// TwinCAT 3 PLC project Untitled1_1
// ProgramVersion: 3.1.4024.0
// libraries:
//   Tc2_MC2, * (Beckhoff Automation GmbH)
//   Tc2_Standard, * (Beckhoff Automation GmbH)
//   Tc2_System, * (Beckhoff Automation GmbH)
//   Tc2_Utilities, * (Beckhoff Automation GmbH)
//   Tc3_IotBase, * (Beckhoff Automation GmbH)
//   Tc3_JsonXml, * (Beckhoff Automation GmbH)
//   Tc3_Module, * (Beckhoff Automation GmbH)
// project tree:
//   DUTs/ E_Mode.TcDUT, E_State.TcDUT, ST_jsoncmd.TcDUT
//   / GlobalTextList.TcGTLO, PlcTask.TcTTO, Visualization Manager.TcVMO (not stored)
//   GVLs/ Comms.TcGVL, E_HomeState.TcDUT, E_LifterState.TcDUT, IO.TcGVL, Slots.TcGVL, ST_Coord.TcDUT, ST_Message.TcDUT
//   POUs/ FBMotion.TcPOU, FB_Lifter.TcPOU, MAIN.TcPOU, Motion.TcPOU, MqttClient.TcPOU, PrgMqttCom.TcPOU
//   VISUs/ Visualization.TcVIS
// real-time tasks:
//   TASK PlcTask: cycle T#10ms, priority 20, ADS port 350
// motion (NC):
//   TASK NC-Task 1 SAF: cycle T#2ms, priority 4, ADS port 501
//   TASK NC-Task 1 SVB: cycle T#10ms, priority 8, ADS port 511
//   AXIS Axis 1 (id 1)
//     Dynamic: Acceleration=322.5, Deceleration=322.5, Jerk=7172.84
//     Velo: SlowManual=10, FastManual=50, Maximum=50
//     OtherSettings: AllowMotionCmdToSlave=true
//     encoder EncType=19
//       EncPara: ScaleFactorNumerator=0.00086, MaxCount=#xffffffff
//     drive DrvType=16
//       DrvPara: MaxCount=#xffffffff, DriveControlDWord=#x00020100
//         Analog: VeloReferenz=50, TorqueSetpointScale=10, ScaleFactorActTorque=0.1
//         TimeComp: TaskDelayCycles=1
//     controller CtrType=1
//       CtrPara: PriorControlFactor=1
//         Observer: BandWidth=20
//   AXIS Axis 2 (id 2)
//     Dynamic: Acceleration=330, Deceleration=330, Jerk=6806.25
//     Velo: SlowManual=10, FastManual=50, Maximum=50
//     OtherSettings: AllowMotionCmdToSlave=true
//     encoder EncType=19
//       EncPara: ScaleFactorNumerator=0.00086, Inverse=true, MaxCount=#xffffffff
//     drive DrvType=16
//       DrvPara: Inverse=true, MaxCount=#xffffffff, DriveControlDWord=#x00020100
//         Analog: VeloReferenz=50, TorqueSetpointScale=10, ScaleFactorActTorque=0.1
//         TimeComp: TaskDelayCycles=1
//     controller CtrType=1
//       CtrPara: PriorControlFactor=1
//         Observer: BandWidth=20
// I/O:
//   DEVICE Device 2 (EtherCAT), AmsNetId 5.81.180.16.3.1
//     Drive 1 (R88D-KN01H-ECT) [R88D-KN01H-ECT G5 Series ServoDrive/Motor]
//     Drive 2 (R88D-KN01H-ECT) [R88D-KN01H-ECT G5 Series ServoDrive/Motor]
//   DEVICE Device 1 (NOV-DP-RAM)
//   DEVICE Device 3 (EtherCAT), AmsNetId 5.81.180.16.4.1
//     Term 1 (EK1200) [EK1200-5000 EtherCAT Power supply (2A E-Bus)]
//       Term 4 (EL1008) [EL1008 8Ch. Dig. Input 24V, 3ms]
//       Term 5 (EL2008) [EL2008 8Ch. Dig. Output 24V, 0.5A]
//       Term 4 (EL9011) [EL9011 End Terminal]
// variable links:
//   NC-Task 1 SAF/Axes/Axis 1 <-> Device 2 (EtherCAT)/Drive 1 (R88D-KN01H-ECT)
//     Drive/Inputs/In/nDataIn1 <-> 258th transmit PDO Mapping/Following error actual value
//     Drive/Inputs/In/nDataIn3[0] <-> 258th transmit PDO Mapping/Torque actual value
//     Drive/Inputs/In/nDcOutputTime <-> InfoData/DcOutputShift
//     Drive/Inputs/In/nState1 <-> 258th transmit PDO Mapping/Statusword
//     Drive/Inputs/In/nState2 <-> 258th transmit PDO Mapping/Statusword @bit 8
//     Drive/Inputs/In/nState4 @bit 1 <-> WcState/InputToggle
//     Drive/Inputs/In/nState4 <-> WcState/WcState
//     Drive/Outputs/Out/nCtrl1 <-> 258th receive PDO Mapping/Controlword
//     Drive/Outputs/Out/nCtrl2 <-> 258th receive PDO Mapping/Controlword @bit 8
//     Drive/Outputs/Out/nDataOut1 <-> 258th receive PDO Mapping/Target position
//     Enc/Inputs/In/nDataIn1 <-> 258th transmit PDO Mapping/Position actual value
//     Enc/Inputs/In/nDataIn3 <-> 258th transmit PDO Mapping/Touch probe pos1 pos value
//     Enc/Inputs/In/nDataIn5 <-> 258th transmit PDO Mapping/Touch probe pos2 pos value
//     Enc/Inputs/In/nDcInputTime <-> InfoData/DcInputShift
//     Enc/Inputs/In/nState4 @bit 1 <-> WcState/InputToggle
//     Enc/Inputs/In/nState4 <-> WcState/WcState
//     Enc/Inputs/In/nState5 <-> 258th transmit PDO Mapping/Touch probe status
//     Enc/Inputs/In/nState6 <-> 258th transmit PDO Mapping/Touch probe status @bit 8
//     Enc/Outputs/Out/nCtrl5 <-> 258th receive PDO Mapping/Touch probe function
//     Enc/Outputs/Out/nCtrl6 <-> 258th receive PDO Mapping/Touch probe function @bit 8
//   NC-Task 1 SAF/Axes/Axis 2 <-> Device 2 (EtherCAT)/Drive 2 (R88D-KN01H-ECT)
//     Drive/Inputs/In/nDataIn1 <-> 258th transmit PDO Mapping/Following error actual value
//     Drive/Inputs/In/nDataIn3[0] <-> 258th transmit PDO Mapping/Torque actual value
//     Drive/Inputs/In/nDcOutputTime <-> InfoData/DcOutputShift
//     Drive/Inputs/In/nState1 <-> 258th transmit PDO Mapping/Statusword
//     Drive/Inputs/In/nState2 <-> 258th transmit PDO Mapping/Statusword @bit 8
//     Drive/Inputs/In/nState4 @bit 1 <-> WcState/InputToggle
//     Drive/Inputs/In/nState4 <-> WcState/WcState
//     Drive/Outputs/Out/nCtrl1 <-> 258th receive PDO Mapping/Controlword
//     Drive/Outputs/Out/nCtrl2 <-> 258th receive PDO Mapping/Controlword @bit 8
//     Drive/Outputs/Out/nDataOut1 <-> 258th receive PDO Mapping/Target position
//     Enc/Inputs/In/nDataIn1 <-> 258th transmit PDO Mapping/Position actual value
//     Enc/Inputs/In/nDataIn3 <-> 258th transmit PDO Mapping/Touch probe pos1 pos value
//     Enc/Inputs/In/nDataIn5 <-> 258th transmit PDO Mapping/Touch probe pos2 pos value
//     Enc/Inputs/In/nDcInputTime <-> InfoData/DcInputShift
//     Enc/Inputs/In/nState4 @bit 1 <-> WcState/InputToggle
//     Enc/Inputs/In/nState4 <-> WcState/WcState
//     Enc/Inputs/In/nState5 <-> 258th transmit PDO Mapping/Touch probe status
//     Enc/Inputs/In/nState6 <-> 258th transmit PDO Mapping/Touch probe status @bit 8
//     Enc/Outputs/Out/nCtrl5 <-> 258th receive PDO Mapping/Touch probe function
//     Enc/Outputs/Out/nCtrl6 <-> 258th receive PDO Mapping/Touch probe function @bit 8
//   Untitled1_1/Untitled1_1 Instance <-> Device 3 (EtherCAT)/Term 1 (EK1200)/Term 4 (EL1008)
//     PlcTask Inputs/IO.Anturi_X_1 <-> Channel 1/Input
//     PlcTask Inputs/IO.Anturi_Y_3 <-> Channel 3/Input
//   Untitled1_1/Untitled1_1 Instance <-> Device 3 (EtherCAT)/Term 1 (EK1200)/Term 5 (EL2008)
//     PlcTask Outputs/IO.Nostin <-> Channel 2/Output
//     PlcTask Outputs/IO.bLifter <-> Channel 5/Output
//   Untitled1_1/Untitled1_1 Instance <-> NC-Task 1 SAF/Axes/Axis 1
//     PlcTask Inputs/Motion.AxisRefX.NcToPlc <-> Outputs/ToPlc
//     PlcTask Outputs/Motion.AxisRefX.PlcToNc <-> Inputs/FromPlc
//   Untitled1_1/Untitled1_1 Instance <-> NC-Task 1 SAF/Axes/Axis 2
//     PlcTask Inputs/Motion.AxisRefY.NcToPlc <-> Outputs/ToPlc
//     PlcTask Outputs/Motion.AxisRefY.PlcToNc <-> Inputs/FromPlc

CONFIGURATION Untitled1_1
    RESOURCE PLC ON TwinCAT3
        TASK PlcTask(INTERVAL := T#10ms, PRIORITY := 20);
        PROGRAM MAIN WITH PlcTask : MAIN;
    END_RESOURCE
END_CONFIGURATION

// ---- DUTs/E_Mode.TcDUT
{attribute 'qualified_only'}
{attribute 'strict'}
TYPE E_Mode :
(
	disabled := 0,
	manual,
	auto
);
END_TYPE

// ---- DUTs/E_State.TcDUT
{attribute 'qualified_only'}
{attribute 'strict'}
TYPE E_State :
(
	inactive := 0,
	initialising,
	homing,
	ready,
	move2pick,
	pick,
	pick2,
	pick3,
	move2place,
	place,
	kotiutusnappi
);
END_TYPE

// ---- DUTs/ST_jsoncmd.TcDUT
TYPE ST_jsoncmd :
STRUCT
	from_slot	:INT;
	to_slot		:INT;
END_STRUCT
END_TYPE

// ---- GVLs/E_HomeState.TcDUT
{attribute 'qualified_only'}
{attribute 'strict'}
TYPE E_HomeState :
(
	Inactive := 0,
	Jog,
	Delay,
	SetPos,
	P2P,
	HomedReady,
	SecondPhase,
	SecondDelay,
	FinalDelay,
	FinalHoming
);
END_TYPE

// ---- GVLs/E_LifterState.TcDUT
{attribute 'qualified_only'}
{attribute 'strict'}
TYPE E_LifterState :
(
	KplEiKyydissa,
	NostoAlas,
	NostoImukuppi,
	NostoYlos,
	LaskuAlas,
	LaskuImukuppi,
	LaskuYlos,
	KplKyydissa
);
END_TYPE

// ---- GVLs/ST_Coord.TcDUT
TYPE ST_Coord :
STRUCT
	x	:LREAL;
	y	:LREAL;
END_STRUCT
END_TYPE

// ---- GVLs/ST_Message.TcDUT
TYPE ST_Message :
STRUCT
	from_slot :INT;
	to_slot	:INT;
END_STRUCT
END_TYPE

// ---- GVLs/Comms.TcGVL
{attribute 'qualified_only'}
VAR_GLOBAL
	bSlotCmd :BOOL;
	stSlotCmd :ST_jsoncmd;
	kotiutusnappi :BOOL;
END_VAR

// ---- GVLs/IO.TcGVL
{attribute 'qualified_only'}
VAR_GLOBAL
	bRA1S AT %I*: BOOL;
	bRA2S AT %I*: BOOL;
	Anturi_X_1 AT %I*: BOOL;
	Anturi_Y_3 AT %I*: BOOL;
	bLifter AT %Q*: BOOL;
	Nostin AT %Q*: BOOL;
	

END_VAR

// ---- GVLs/Slots.TcGVL
{attribute 'qualified_only'}
VAR_GLOBAL
	Coords: ARRAY[0..10] OF ST_Coord := [(x := 10, y := 10), (x := 150, y := 10), (x := 250, y := 10), (x := 333.33, y := 41.67), (x := 0, y := 0), (x := 200, y := 125), (x := 333.33, y := 125), (x := 66.667, y := 208.33), (x := 200, y := 208.33), (x := 333.33, y := 208.33), (x := 160, y := 410)];
END_VAR

// ---- POUs/MAIN.TcPOU
PROGRAM MAIN
VAR
END_VAR

Motion();

//PrgMqttCom();

END_PROGRAM

// ---- POUs/Motion.TcPOU
PROGRAM Motion

VAR
	
		

	X: FBMotion;
	Y: FBMotion;  
	AxisRefX: AXIS_REF;
	AxisRefY: AXIS_REF;
	ManualMove: BOOL;
	rTarget_Y: LREAL;
	rTarget_X: LREAL;
	PowerOffStop: BOOL;
	PowerOn: BOOL;
	Reset_X: BOOL;
	Reset_Y: BOOL;
	FindHome: BOOL;
	ManualSlotMove: BOOL;
	SlotVariableY: INT;
	SlotVariableX: INT;
	fbLifter: FB_Lifter;
	Nosto: BOOL;
	Lasku: BOOL;
	eMode: E_Mode := E_MODE.manual;
	eState: E_State;
	AutoInit: BOOL := FALSE;
	tonNostonLaskuDelay: TON := (PT := TIME#1s0ms);
	tonNostonNostoDelay: TON := (PT := TIME#1S0MS);
	tonLaskunLaskuDelay: TON := (PT:= TIME#1S0MS);
	tonXDelayEnnenYP2P: TON := (PT:= TIME#100MS);
	DelayStartNostonLasku: BOOL;
	DelayStartNostonNosto: BOOL;
	DelayStartLaskunLasku: BOOL;
	DelayStartXDelayEnnenYP2P: BOOL;
END_VAR

//X-akseli
X(AxisRef:= AxisRefX, bHomeCalibrationCam:=(IO.Anturi_X_1));

//Y-akseli
Y(AxisRef:= AxisRefY, bHomeCalibrationCam:=(IO.Anturi_Y_3));

//fbLifter();
//IO.bLifter := fbLifter.bLifter;
//IO.Imukuppi := fbLifter.bImukuppi;

tonNostonLaskuDelay(IN:= DelayStartNostonLasku);
tonNostonNostoDelay(IN:= DelayStartNostonNosto);
tonLaskunLaskuDelay(IN:= DelayStartLaskunLasku);
tonXDelayEnnenYP2P(IN:= DelayStartXDelayEnnenYP2P);

CASE eMode OF
	E_Mode.manual:		
		IF ManualMove THEN
			Y.P2P(rTarget_Y);
			X.P2P(rTarget_X);
			ManualMove := FALSE;
		END_IF
		
		IF ManualSlotMove THEN
			Y.P2P(Slots.Coords[SlotVariableY].y);
			X.P2P(Slots.Coords[SlotVariableX].x);
			ManualSlotMove := FALSE;
		END_IF
		
		IF Reset_X THEN
			X.Reset();
			Reset_X := FALSE;
		END_IF
		
		IF Reset_Y THEN
			Y.Reset();
			Reset_Y := FALSE;
		END_IF
		
		
		IF PowerOffStop THEN
			X.PowerOff();
			Y.PowerOff();
			PowerOffStop := FALSE;
		END_IF
		
		IF PowerOn THEN
			X.PowerOn();
			Y.PowerOn();
			PowerOn := FALSE;
		END_IF
		
		IF FindHome THEN
			X.FindHome();
			IF X.bHomed THEN
				Y.FindHome();
				FindHome := FALSE;
			END_IF
			
		END_IF
		
		IF Nosto THEN
			fbLifter.KplNosto();
			Nosto := FALSE;
		END_IF
		
		IF Lasku THEN
			fbLifter.KplLasku();
			Lasku := FALSE;
		END_IF
	
	E_Mode.auto:
		CASE eState OF
			E_State.inactive:
				IF AutoInit THEN
					AutoInit:= FALSE;
					X.PowerOn();
					Y.PowerOn();
					eState := E_state.initialising;
				END_IF
	
			E_State.initialising:
				IF X.bPowerStatus AND Y.bPowerStatus THEN
					X.FindHome();
					//Y.FindHome();
					eState := E_state.homing;
				END_IF
			
			E_State.homing:
				IF X.bHomed  THEN //AND Y.bHomed THEN
					Y.FindHome();		
					IF Y.bHomed THEN
						eState := E_state.ready;	
					END_IF		
				END_IF
				
			E_State.ready:
				IF Comms.bSlotCmd THEN
					Comms.bSlotCmd := FALSE;
					X.P2P(Slots.Coords[Comms.stSlotCmd.from_slot].x);
					Y.P2P(Slots.Coords[Comms.stSlotCmd.from_slot].y);
					eState := E_state.move2pick;
				ELSIF Comms.kotiutusnappi THEN
					Comms.kotiutusnappi := FALSE;
					Y.P2P(0.0);
					X.P2P(0.0);
					eState := E_state.kotiutusnappi;
				END_IF
				
			E_State.move2pick:
				IF X.bP2P_Ready AND Y.bP2P_Ready THEN
					// fbLifter.KplNosto();
					IO.Nostin := TRUE;
					tonNostonLaskuDelay.PT := T#1S;
					DelayStartNostonLasku := TRUE;
					IF tonNostonLaskuDelay.Q THEN
						DelayStartNostonLasku := FALSE;
						Y.P2P(AxisRefY.NcToPlc.ActPos + 100);
						eState := E_state.pick;
					END_IF
				END_IF
				
			E_State.pick:
				IF Y.bP2P_Ready THEN
					IO.Nostin := FALSE;
					tonNostonNostoDelay.PT := T#1S;
					DelayStartNostonNosto := TRUE;
					IF tonNostonNostoDelay.Q THEN
						DelayStartNostonNosto := FALSE;
						Y.P2P(AxisRefY.NcToPlc.ActPos - 100);
						eState := E_state.pick2;
					END_IF
				END_IF;
					
			E_State.pick2:
				IF Y.bP2P_Ready THEN
					X.P2P(Slots.Coords[Comms.stSlotCmd.to_slot].x);
					eState := E_state.pick3;
				END_IF
				
			E_State.pick3:
				IF X.bP2P_Ready THEN
					Y.P2P(Slots.Coords[Comms.stSlotCmd.to_slot].y + 100);
					eState := E_state.move2place;
				END_IF
				
			E_State.move2place:
				IF X.bP2P_Ready AND Y.bP2P_Ready THEN
					// fbLifter.KplLasku();
					IO.Nostin := TRUE;
					tonLaskunLaskuDelay.PT := T#1S;
					DelayStartLaskunLasku := TRUE;
					IF tonLaskunLaskuDelay.Q THEN
						DelayStartLaskunLasku := FALSE;
						Y.P2P(AxisRefY.NcToPlc.ActPos - 100);
						eState := E_state.place;
					END_IF
				END_IF
				
			E_State.place:
				IF X.bP2P_Ready AND Y.bP2P_Ready THEN
					IO.Nostin := FALSE;
					eState := E_state.ready;
				END_IF;

			E_State.kotiutusnappi:
				IF X.bP2P_Ready AND Y.bP2P_Ready THEN
					eState := E_state.ready;
				END_IF;
		END_CASE
END_CASE

END_PROGRAM

// ---- POUs/FBMotion.TcPOU
FUNCTION_BLOCK FBMotion
VAR
	AxisPower: MC_Power;
	AxisMoveabsolute: MC_MoveAbsolute;
	AxisHome: MC_Home;
	AxisReset: MC_Reset;
	bHomeExec: BOOL;
	bMoveExec: BOOL;
	MoveToHome: LREAL;
	rVelocity: LREAL := 30;
	rAcceleration: LREAL := 1000;
	rDeceleration: LREAL := 1000;
	rJerk: LREAL := 1000;
	HomeOptions: ST_HomingOptions;
	MoveOptions: ST_MoveOptions;
	PowerOptions: ST_PowerOptions;
	PowerBufferMode: MC_BufferMode;
	HomingMode: MC_HomingMode;
	HomeBufferMode: MC_BufferMode;
	MoveBufferMove: MC_BufferMode;
	MoveBufferMode: MC_BufferMode;
	nDistanceToTarget: INT;
	rDistanceToTarget: LREAL;
	bResetExec: BOOL;
	luku: INT;
END_VAR
VAR_OUTPUT
	bPowerStatus: BOOL;
END_VAR
VAR
	AxisJog: MC_Jog;
	bJogForward: BOOL;
	bJogBackward: BOOL;
	JogMode: E_JogMode := E_JOGMODE.MC_JOGMODE_CONTINOUS;
	rJogVelocity: LREAL := 30;
	rJogAcceleration: LREAL := 1000;
	rJogDeceleration: LREAL := 1000;
	rJogJerk: LREAL := 1000;
	rJogMoveToPos: LREAL;
	rMoveToPos: LREAL;
	eHomeState: E_HomeState;
	bHomeCmd: BOOL;
	tonHomeDelay: TON := (PT := TIME#2S0MS);
	tonSecondDelay: TON := (PT := TIME#500MS);
	tonFinalDelay: TON := (PT := TIME#1S0MS);
	fbSetPosition: MC_SetPosition;
	bSetPosition: BOOL;
	rSetPosition: LREAL := 0;
	SetPos: ST_McOutputs;
END_VAR
VAR_INPUT
	bHomeCalibrationCam: BOOL;
END_VAR
VAR
	bPowerEnable: BOOL := TRUE;
END_VAR
VAR_IN_OUT
	AxisRef: AXIS_REF;
END_VAR
VAR
	MoveOut: ST_McOutputs;
	HomeOut: ST_McOutputs;
	PowerOut: ST_McOutputs;
	JogOut: ST_McOutputs;
	ResetOut: ST_McOutputs;
END_VAR

VAR_OUTPUT
	bHomed: BOOL;
	bP2P_Ready: BOOL;
END_VAR

AxisPower(
	Axis:= AxisRef, 
	Enable:= bPowerEnable, 
	Enable_Positive:= TRUE, 
	Enable_Negative:= TRUE, 
	Override:= 100.0, 
	BufferMode:= PowerBufferMode, 
	Options:= PowerOptions, 
	Status=> bPowerStatus, 		
	Busy=> PowerOut.Busy,        
	Active=> PowerOut.Active,      
	Error=> PowerOut.Error,       
	ErrorID=> PowerOut.ErrorID);    

(*	
AxisHome(
	Axis:= AxisRef, 
	Execute:= bHomeExec, 
	Position:= MoveToHome, 
	HomingMode:= HomingMode, 
	BufferMode:= HomeBufferMode, 
	Options:= HomeOptions, 
	bCalibrationCam:= bHomeCalibrationCam, 
	Done=> 				HomeOut.Done, 
	Busy=> 				HomeOut.Busy, 
	Active=> 			HomeOut.Active, 
	CommandAborted=> 	HomeOut.CommandAborted, 
	Error=> 			HomeOut.Error, 
	ErrorID=> 			HomeOut.ErrorID);
	*)

AxisReset(
	Axis:= AxisRef, 
	Execute:= bResetExec, 
	Done=> ResetOut.Done, 
	Busy=> ResetOut.Busy, 
	Error=> ResetOut.Error, 
	ErrorID=> ResetOut.ErrorID);

//bResetExec := FALSE;
	
AxisMoveabsolute(
	Axis:= AxisRef, 
	Execute:= bMoveExec, 
	Position:= rMoveToPos, 
	Velocity:= rVelocity, 
	Acceleration:= rAcceleration, 
	Deceleration:= rDeceleration, 
	Jerk:= rJerk, 
	BufferMode:= MoveBufferMode, 
	Options:= MoveOptions, 
	Done=> 				MoveOut.Done, 
	Busy=> 				MoveOut.Busy, 
	Active=> 			MoveOut.Active, 
	CommandAborted=> 	MoveOut.CommandAborted, 
	Error=> 			MoveOut.Error, 
	ErrorID=> 			MoveOut.ErrorID);
	
bMoveExec := FALSE;

AxisJog(
	Axis:= AxisRef , 
	JogForward:= bJogForward, 
	JogBackwards:= bJogBackward, 
	Mode:= JogMode, 
	Position:= rJogMoveToPos, 
	Velocity:= rJogVelocity, 
	Acceleration:= rJogAcceleration, 
	Deceleration:= rJogDeceleration, 
	Jerk:= rJogJerk, 
	Done=> JogOut.Done, 
	Busy=> JogOut.Busy, 
	Active=> JogOut.Active, 
	CommandAborted=> JogOut.CommandAborted, 
	Error=> JogOut.Error, 
	ErrorID=> JogOut.ErrorID);

fbSetPosition(
	Axis:= AxisRef, 
	Execute:= bSetPosition, 
	Position:= rSetPosition, 
	Mode:= FALSE, 
	Options:= , 
	Done=> SetPos.Done, 
	Busy=> SetPos.Busy, 
	Error=> SetPos.Error, 
	ErrorID=> SetPos.ErrorID);

tonHomeDelay(IN:= eHomeState = E_HomeState.Delay);
tonSecondDelay(IN:= eHomeState = E_HomeState.SecondDelay);	
tonFinalDelay(IN:= eHomeState = E_HomeState.FinalDelay);		
bHomed := FALSE;



CASE eHomeState OF
	E_HomeState.Inactive:
		 IF bHomeCmd THEN
			 eHomeState := E_HomeState.Jog;
		 END_IF
	E_HomeState.Jog:
		bJogBackward:=TRUE;
		IF bHomeCalibrationCam THEN
			bJogBackward:=FALSE;
			eHomeState := E_HomeState.Delay;
		END_IF
//	E_HomeState.Delay:
//		 IF tonHomeDelay.Q THEN
//			 eHomeState := E_HomeState.SetPos;
//		 END_IF		
//// homing lisä
	E_HomeState.Delay:
		IF tonHomeDelay.Q THEN
			eHomeState := E_HomeState.SecondPhase;
		END_IF
	E_HomeState.SecondPhase:
		IF bHomeCalibrationCam THEN
			bJogForward:= TRUE;
			eHomeState := E_HomeState.SecondDelay;
		END_IF
	E_HomeState.SecondDelay:
		IF tonSecondDelay.Q THEN
			bJogForward:= FALSE;
			eHomeState := E_HomeState.FinalHoming;
		END_IF
	E_HomeState.FinalHoming:
		rJogVelocity := 2;
		bJogBackward:= TRUE;
		IF bHomeCalibrationCam THEN
			bJogBackward:= FALSE;
			rJogVelocity := 30;
			eHomeState:= E_HomeState.FinalDelay;
		END_IF
	E_HomeState.FinalDelay:
		IF tonFinalDelay.Q THEN
			eHomeState := E_HomeState.SetPos;
		END_IF
////////
	E_HomeState.SetPos:
		bSetPosition := TRUE;
		IF SetPos.Done THEN
			bSetPosition := FALSE;
			eHomeState := E_HomeState.HomedReady;
		END_IF	
	(*
	E_HomeState.P2P:
		P2P(0);
		IF MoveOut.Done THEN
			eHomeState := E_HomeState.HomedReady;
		END_IF
	*)
	E_HomeState.HomedReady:
		bHomed := TRUE;
			
END_CASE

 bHomeCmd := FALSE;
 
 rDistanceToTarget := ABS(AxisRef.NcToPlc.ActPos - rMoveToPos);
 bP2P_Ready := rDistanceToTarget < 0.1 AND bHomed;

METHOD FindHome : BOOL
VAR_INPUT
END_VAR
IF eHomeState = E_HomeState.Inactive THEN
	bHomeCmd := TRUE;
	FindHome := TRUE;
ELSE
	FindHome := FALSE;
END_IF
END_METHOD

METHOD P2P : BOOL
VAR_INPUT
	TargetPos: LREAL;
END_VAR


IF bPowerStatus THEN
	rMoveToPos := TargetPos;
	bMoveExec := TRUE;
	P2P := TRUE;
	bP2P_Ready := FALSE;
ELSE
	P2P := FALSE;
END_IF
END_METHOD

METHOD PowerOff : BOOL
VAR_INPUT
END_VAR
bPowerEnable := FALSE;
END_METHOD

METHOD PowerOn : BOOL
VAR_INPUT
END_VAR
bPowerEnable := TRUE;
END_METHOD

METHOD Reset : BOOL
VAR_INPUT
END_VAR
bResetExec := TRUE;
END_METHOD

END_FUNCTION_BLOCK

// ---- POUs/FB_Lifter.TcPOU
FUNCTION_BLOCK FB_Lifter
VAR_OUTPUT
	bLifter: BOOL;
	bImukuppi: BOOL;
END_VAR
VAR
	DelayStart: BOOL;
	tonImukuppiDelay: TON := (PT := TIME#2s0ms);
	LifterState: E_LifterState;
	NostoCMD: BOOL;
	bKplKyydissa: BOOL;
	LaskuCMD: BOOL;
END_VAR
VAR_OUTPUT
	Ready: BOOL;
END_VAR


tonImukuppiDelay(IN := DelayStart);



CASE LifterState OF
	
	E_LifterState.KplEiKyydissa:
		Ready := TRUE;
		IF NostoCMD = TRUE THEN
			LifterState := E_LifterState.NostoAlas;
			Ready := FALSE;
		END_IF
	
	E_LifterState.NostoAlas:
		Ready := FALSE;
		bLifter := TRUE;
		tonImukuppiDelay.PT := T#1S;
		DelayStart := TRUE;
		IF tonImukuppiDelay.Q THEN
			DelayStart := FALSE;
			LifterState := E_LifterState.NostoImukuppi;
		END_IF
	
	E_LifterState.NostoImukuppi:
		bImukuppi := TRUE;
		bLifter := TRUE;
		tonImukuppiDelay.PT := T#2S;
		DelayStart := TRUE;
		IF tonImukuppiDelay.Q THEN
			DelayStart := FALSE;
			LifterState := E_LifterState.NostoYlos;
		END_IF
	
	E_LifterState.NostoYlos:
		bLifter := FALSE;
		tonImukuppiDelay.PT := T#2S;
		DelayStart := TRUE;
		IF tonImukuppiDelay.Q THEN
			DelayStart := FALSE;
			LifterState := E_LifterState.KplKyydissa;
		END_IF	
	
	/////////////////////
	
	E_LifterState.KplKyydissa:
		Ready := TRUE;
		bKplKyydissa :=TRUE;
		IF LaskuCMD = TRUE THEN
			Ready := FALSE;
			LifterState := E_LifterState.LaskuAlas;
		END_IF
	
	/////////////////////////
	
	
	E_LifterState.LaskuAlas:
		Ready := FALSE;
		bLifter := TRUE;
		tonImukuppiDelay.PT := T#1S;
		DelayStart := TRUE;
		IF tonImukuppiDelay.Q THEN
			DelayStart := FALSE;
			LifterState := E_LifterState.LaskuImukuppi;
		END_IF
	
	E_LifterState.LaskuImukuppi:
		bImukuppi := FALSE;
		bLifter := TRUE;
		tonImukuppiDelay.PT := T#2S;
		DelayStart := TRUE;
		IF tonImukuppiDelay.Q THEN
			DelayStart := FALSE;
			LifterState := E_LifterState.LaskuYlos;
		END_IF
	
	E_LifterState.LaskuYlos:
		bLifter := FALSE;
		tonImukuppiDelay.PT := T#2S;
		DelayStart := TRUE;
		IF tonImukuppiDelay.Q THEN
			DelayStart := FALSE;
			LifterState := E_LifterState.KplEiKyydissa;
		END_IF	
	
END_CASE

LaskuCMD := FALSE;
NostoCMD := FALSE;

METHOD KplLasku : BOOL
VAR_INPUT
END_VAR
LaskuCMD := TRUE;
END_METHOD

METHOD KplNosto : BOOL
NostoCMD := TRUE;
END_METHOD

END_FUNCTION_BLOCK

// ---- POUs/MqttClient.TcPOU
FUNCTION MqttClient : FB_IotMqtt5Client
PROGRAM PrgMqttCom
VAR
    fbMqttClient    : FB_IotMqttClient;
    bSetParameter   : BOOL := TRUE;
    bConnect        : BOOL := TRUE;
END_VAR

// NETWORK 1

END_FUNCTION

// ---- POUs/PrgMqttCom.TcPOU
PROGRAM PrgMqttCom
VAR
	fbMqttClient    : FB_IotMqttClient;
    bSetParameter   : BOOL := TRUE;
    bConnect        : BOOL := TRUE;
	
	(* published message *)
    sTopicPub   : STRING(255) := 'plc2pc';
    sPayloadPub : STRING(255);
    i : UDINT;
    fbTimer : TON := (PT:=T#10S);
	
	(* received message *)
    bSubscribed    : BOOL;
    sTopicSub      : STRING(255) := 'pc2plc';
    {attribute 'TcEncoding':='UTF-8'}
    sTopicRcv      : STRING(255);
    {attribute 'TcEncoding':='UTF-8'}
    sPayloadRcv    : STRING(255);
    fbMessageQueue : FB_IotMqttMessageQueue;
    fbMessage      : FB_IotMqttMessage;
	
	  fbJson     : FB_JsonDomParser;
	  jsonDoc    : SJsonValue;
	  jsonProp   : SJsonValue;
	  jsonValue  : SJsonValue;
	  bHasMember : BOOL;
	  
	   sMessage   : STRING(255) := '{"serialNumber":"G030PT028191AC4R","batteryVoltage":"1547mV","clickType":"SINGLE"}';
	  
	  stReceivedData : ST_jsoncmd;
	
	a_pos: INT := 1;
	b_pos: INT := 1;
	bias: INT:=4;
	a_char: STRING(255);
	b_char: STRING(255);
	
	a_len: INT :=1;
	b_len: INT :=1;
END_VAR

IF bSetParameter THEN
    bSetParameter               := FALSE;
    fbMqttClient.sHostName      := 'localhost';
    fbMqttClient.nHostPort      := 1883;
    fbMqttClient.sClientId      := 'varastoplc'; 
    fbMqttClient.sTopicPrefix   := ''; 
//    fbMqttClient.nKeepAlive     := 60; 
    fbMqttClient.sUserName      := 'admin';
    fbMqttClient.sUserPassword  := 'tietotekniikka3'; 
//  fbMqttClient.stWill         := ; 
//  fbMqttClient.stTLS          := ;
    fbMqttClient.ipMessageQueue := fbMessageQueue;
END_IF

fbMqttClient.Execute(bConnect);

IF fbMqttClient.bConnected THEN
    IF NOT bSubscribed THEN
        bSubscribed := fbMqttClient.Subscribe(sTopic:=sTopicSub, eQoS:=TcIotMqttQos.AtMostOnceDelivery);
    END_IF
    fbTimer(IN:=TRUE);
    IF fbTimer.Q THEN // publish new payload every second
        fbTimer(IN:=FALSE);
        i := i + 1;
        sPayloadPub := CONCAT('MyMessage', TO_STRING(i));
        fbMqttClient.Publish(    sTopic:= sTopicPub, 
                                pPayload:= ADR(sPayloadPub), nPayloadSize:= LEN2(ADR(sPayloadPub))+1, 
                                eQoS:= TcIotMqttQos.AtMostOnceDelivery, bRetain:= FALSE, bQueue:= FALSE );
    END_IF
END_IF

IF fbMessageQueue.nQueuedMessages > 0 THEN
    IF fbMessageQueue.Dequeue(fbMessage:=fbMessage) THEN
        fbMessage.GetTopic(pTopic:=ADR(sTopicRcv), nTopicSize:=SIZEOF(sTopicRcv) );
        fbMessage.GetPayload(pPayload:=ADR(sPayloadRcv), nPayloadSize:=SIZEOF(sPayloadRcv), bSetNullTermination:=TRUE);
    END_IF
END_IF

(* Hieman hämyinen quick'n'dirty parseri - Tukee vain yhden tai kahden merkin mittaisia slotteja *)

a_pos := FIND(sPayloadRcv,'A');
b_pos := FIND(sPayloadRcv,'B');

// If messgae has both values
IF a_pos > 0 AND b_pos > 0 THEN
	IF MID(sPayloadRcv,1,a_pos + bias + 1) = ','THEN
		a_len := 1;
	ELSE
		a_len := 2;
	END_IF
	
	IF MID(sPayloadRcv,1,b_pos + bias + 1) = '}' THEN
		b_len := 1;
	ELSE
		b_len := 2;
	END_IF
	
	a_char := MID(sPayloadRcv,a_len,a_pos + bias);
	b_char := MID(sPayloadRcv,b_len,b_pos + bias);
	
	Comms.stSlotCmd.from_slot := STRING_TO_INT(a_char);
	Comms.stSlotCmd.to_slot := STRING_TO_INT(b_char);
	Comms.bSlotCmd := TRUE;
	
	sPayloadRcv := '';
ELSE
	Comms.bSlotCmd := FALSE;
END_IF



(* Something fuzzy with json chars
//jsonDoc := fbJson.ParseDocument(sPayloadRcv);
jsonDoc := fbJson.ParseDocument(sMessage);

jsonProp := fbJson.FindMember(jsonDoc, 'from_slot');
IF (jsonProp <> 0) THEN
  stReceivedData.from_slot := DINT_TO_INT(fbJson.GetInt(jsonProp));
END_IF

jsonProp := fbJson.FindMember(jsonDoc, 'to_slot');
IF (jsonProp <> 0) THEN
  stReceivedData.to_slot := DINT_TO_INT(fbJson.GetInt(jsonProp));
END_IF

*)

END_PROGRAM

// ---- GlobalTextList.TcGTLO
TEXTLIST GlobalTextList
  708 = 'Home'
  457 = 'Siirrä'
  783 = 'TEE'
END_TEXTLIST

// ---- VISUs/Visualization.TcVIS
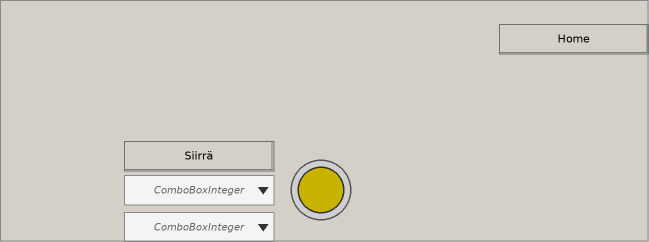
VISUALIZATION Visualization  // 649x242
    Button (499,24 150x30), "Home"
        tap Comms.kotiutusnappi
    Lamp1 (286,155 70x70), style: Lamp-Lamp1-Yellow
    ComboBoxInteger (124,212 150x30), variable: Comms.stSlotCmd.to_slot
    Button (124,141 150x30), "Siirrä"
        tap Comms.bSlotCmd
    ComboBoxInteger (124,175 150x30), variable: Comms.stSlotCmd.from_slot
END_VISUALIZATION
